		MoveL Tr_meulage_motif_1_P35,[12.5,500,0,0],z0,Tool \wobj:=Wobj_Part_0;
		MoveL Tr_meulage_motif_1_P36,[12.5,500,0,0],z0,Tool \wobj:=Wobj_Part_0;
		MoveL Tr_meulage_motif_1_P37,[12.5,500,0,0],z0,Tool \wobj:=Wobj_Part_0;
		MoveL Tr_meulage_motif_1_P38,[12.5,500,0,0],z0,Tool \wobj:=Wobj_Part_0;
		MoveL Tr_meulage_motif_1_P39,[12.5,500,0,0],z0,Tool \wobj:=Wobj_Part_0;
		MoveL Tr_meulage_motif_1_P40,[12.5,500,0,0],z0,Tool \wobj:=Wobj_Part_0;
		MoveL Tr_meulage_motif_1_P41,[12.5,500,0,0],z0,Tool \wobj:=Wobj_Part_0;
		MoveL Tr_meulage_motif_1_P42,[12.5,500,0,0],z0,Tool \wobj:=Wobj_Part_0;
		MoveL Tr_meulage_motif_1_P43,[12.5,500,0,0],z0,Tool \wobj:=Wobj_Part_0;
		MoveL Tr_meulage_motif_1_P44,[12.5,500,0,0],z0,Tool \wobj:=Wobj_Part_0;
		MoveL Tr_meulage_motif_1_P45,[12.5,500,0,0],z0,Tool \wobj:=Wobj_Part_0;
		MoveL Tr_meulage_motif_1_P46,[12.5,500,0,0],z0,Tool \wobj:=Wobj_Part_0;
		MoveL Tr_meulage_motif_1_P47,[12.5,500,0,0],z0,Tool \wobj:=Wobj_Part_0;
		MoveL Tr_meulage_motif_1_P48,[12.5,500,0,0],z0,Tool \wobj:=Wobj_Part_0;
		MoveL Tr_meulage_motif_1_P49,[12.5,500,0,0],z0,Tool \wobj:=Wobj_Part_0;
		MoveL Tr_meulage_motif_1_P50,[12.5,500,0,0],z0,Tool \wobj:=Wobj_Part_0;
		MoveL Tr_meulage_motif_1_P51,[12.5,500,0,0],z0,Tool \wobj:=Wobj_Part_0;
		MoveL Tr_meulage_motif_1_P52,[12.5,500,0,0],z0,Tool \wobj:=Wobj_Part_0;
		MoveL Tr_meulage_motif_1_P53,[12.5,500,0,0],z0,Tool \wobj:=Wobj_Part_0;
		MoveL Tr_meulage_motif_1_P54,[12.5,500,0,0],z0,Tool \wobj:=Wobj_Part_0;
		MoveL Tr_meulage_motif_1_P55,[12.5,500,0,0],z0,Tool \wobj:=Wobj_Part_0;
		MoveL Tr_meulage_motif_1_P56,[12.5,500,0,0],z0,Tool \wobj:=Wobj_Part_0;
		MoveL Tr_meulage_motif_1_P57,[12.5,500,0,0],z0,Tool \wobj:=Wobj_Part_0;
		MoveL Tr_meulage_motif_1_P58,[12.5,500,0,0],z0,Tool \wobj:=Wobj_Part_0;
		MoveL Tr_meulage_motif_1_P59,[12.5,500,0,0],z0,Tool \wobj:=Wobj_Part_0;
		MoveL Tr_meulage_motif_1_P60,[12.5,500,0,0],z0,Tool \wobj:=Wobj_Part_0;
		MoveL Tr_meulage_motif_1_P61,[12.5,500,0,0],z0,Tool \wobj:=Wobj_Part_0;
		MoveL Tr_meulage_motif_1_P62,[12.5,500,0,0],z0,Tool \wobj:=Wobj_Part_0;
		MoveL Tr_meulage_motif_1_P63,[12.5,500,0,0],z0,Tool \wobj:=Wobj_Part_0;
		MoveL Tr_meulage_motif_1_P64,[12.5,500,0,0],z0,Tool \wobj:=Wobj_Part_0;
		MoveL Tr_meulage_motif_1_P65,[12.5,500,0,0],z0,Tool \wobj:=Wobj_Part_0;
		MoveL Tr_meulage_motif_1_P66,[12.5,500,0,0],z0,Tool \wobj:=Wobj_Part_0;
		MoveL Tr_meulage_motif_1_P67,[12.5,500,0,0],z0,Tool \wobj:=Wobj_Part_0;
		MoveL Tr_meulage_motif_1_P68,[12.5,500,0,0],z0,Tool \wobj:=Wobj_Part_0;
		MoveL Tr_meulage_motif_1_P69,[12.5,500,0,0],z0,Tool \wobj:=Wobj_Part_0;
		MoveL Tr_meulage_motif_1_P70,[12.5,500,0,0],z0,Tool \wobj:=Wobj_Part_0;
		MoveL Tr_meulage_motif_1_P71,[12.5,500,0,0],z0,Tool \wobj:=Wobj_Part_0;
		MoveL Tr_meulage_motif_1_P72,[12.5,500,0,0],z0,Tool \wobj:=Wobj_Part_0;
		MoveL Tr_meulage_motif_1_P73,[12.5,500,0,0],z0,Tool \wobj:=Wobj_Part_0;
		MoveL Tr_meulage_motif_1_P74,[12.5,500,0,0],z0,Tool \wobj:=Wobj_Part_0;
		MoveL Tr_meulage_motif_1_P75,[12.5,500,0,0],z0,Tool \wobj:=Wobj_Part_0;
		MoveL Tr_meulage_motif_1_P76,[12.5,500,0,0],z0,Tool \wobj:=Wobj_Part_0;
		MoveL Tr_meulage_motif_1_P77,[12.5,500,0,0],z0,Tool \wobj:=Wobj_Part_0;
		MoveL Tr_meulage_motif_1_P78,[12.5,500,0,0],z0,Tool \wobj:=Wobj_Part_0;
		MoveL Tr_meulage_motif_1_P79,[12.5,500,0,0],z0,Tool \wobj:=Wobj_Part_0;
		MoveL Tr_meulage_motif_1_P80,[12.5,500,0,0],z0,Tool \wobj:=Wobj_Part_0;
		MoveL Tr_meulage_motif_1_P81,[12.5,500,0,0],z0,Tool \wobj:=Wobj_Part_0;
		MoveL Tr_meulage_motif_1_P82,[12.5,500,0,0],z0,Tool \wobj:=Wobj_Part_0;
		MoveL Tr_meulage_motif_1_P83,[12.5,500,0,0],z0,Tool \wobj:=Wobj_Part_0;
		MoveL Tr_meulage_motif_1_P84,[12.5,500,0,0],z0,Tool \wobj:=Wobj_Part_0;
		MoveL Tr_meulage_motif_1_P85,[12.5,500,0,0],z0,Tool \wobj:=Wobj_Part_0;
		MoveL Tr_meulage_motif_1_P86,[12.5,500,0,0],z0,Tool \wobj:=Wobj_Part_0;
		MoveL Tr_meulage_motif_1_P87,[12.5,500,0,0],z0,Tool \wobj:=Wobj_Part_0;
		MoveL Tr_meulage_motif_1_P88,[12.5,500,0,0],z0,Tool \wobj:=Wobj_Part_0;
		MoveL Tr_meulage_motif_1_P89,[12.5,500,0,0],z0,Tool \wobj:=Wobj_Part_0;
		MoveL Tr_meulage_motif_1_P90,[12.5,500,0,0],z0,Tool \wobj:=Wobj_Part_0;
		MoveL Tr_meulage_motif_1_P91,[12.5,500,0,0],z0,Tool \wobj:=Wobj_Part_0;
		MoveL Tr_meulage_motif_1_P92,[12.5,500,0,0],z0,Tool \wobj:=Wobj_Part_0;
		MoveL Tr_meulage_motif_1_P93,[12.5,500,0,0],z0,Tool \wobj:=Wobj_Part_0;
		MoveL Tr_meulage_motif_1_P94,[12.5,500,0,0],z0,Tool \wobj:=Wobj_Part_0;
		MoveL Tr_meulage_motif_1_P95,[12.5,500,0,0],z0,Tool \wobj:=Wobj_Part_0;
		MoveL Tr_meulage_motif_1_P96,[12.5,500,0,0],z0,Tool \wobj:=Wobj_Part_0;
		MoveL Tr_meulage_motif_1_P97,[12.5,500,0,0],z0,Tool \wobj:=Wobj_Part_0;
		MoveL Tr_meulage_motif_1_P98,[12.5,500,0,0],z0,Tool \wobj:=Wobj_Part_0;
		MoveL Tr_meulage_motif_1_P99,[12.5,500,0,0],z0,Tool \wobj:=Wobj_Part_0;
		MoveL Tr_meulage_motif_1_P100,[12.5,500,0,0],z0,Tool \wobj:=Wobj_Part_0;
		MoveL Tr_meulage_motif_1_P101,[12.5,500,0,0],z0,Tool \wobj:=Wobj_Part_0;
		MoveL Tr_meulage_motif_1_P102,[12.5,500,0,0],z0,Tool \wobj:=Wobj_Part_0;
		MoveL Tr_meulage_motif_1_P103,[12.5,500,0,0],z0,Tool \wobj:=Wobj_Part_0;
		MoveL Tr_meulage_motif_1_P104,[12.5,500,0,0],z0,Tool \wobj:=Wobj_Part_0;
		MoveL Tr_meulage_motif_1_P105,[12.5,500,0,0],z0,Tool \wobj:=Wobj_Part_0;
		MoveL Tr_meulage_motif_1_P106,[12.5,500,0,0],z0,Tool \wobj:=Wobj_Part_0;
		MoveL Tr_meulage_motif_1_P107,[12.5,500,0,0],z0,Tool \wobj:=Wobj_Part_0;
		MoveL Tr_meulage_motif_1_P108,[12.5,500,0,0],z0,Tool \wobj:=Wobj_Part_0;
		MoveL Tr_meulage_motif_1_P109,[12.5,500,0,0],z0,Tool \wobj:=Wobj_Part_0;
		MoveL Tr_meulage_motif_1_P110,[12.5,500,0,0],z0,Tool \wobj:=Wobj_Part_0;
		MoveL Tr_meulage_motif_1_P111,[12.5,500,0,0],z0,Tool \wobj:=Wobj_Part_0;
		MoveL Tr_meulage_motif_1_P112,[12.5,500,0,0],z0,Tool \wobj:=Wobj_Part_0;
		MoveL Tr_meulage_motif_1_P113,[12.5,500,0,0],z0,Tool \wobj:=Wobj_Part_0;
		MoveL Tr_meulage_motif_1_P114,[12.5,500,0,0],z0,Tool \wobj:=Wobj_Part_0;
		MoveL Tr_meulage_motif_1_P115,[12.5,500,0,0],z0,Tool \wobj:=Wobj_Part_0;
		MoveJ Tr_meulage_motif_1_degg1,V500,Z0,Tool,\Wobj:=Wobj_Part_0;
		MoveJ Tr_meulage_motif_1_degg2,V2000,Z100,Tool,\Wobj:=Wobj_Part_0;
	ENDPROC
	LOCAL PROC Tr_meulage_motif_2()
		!!Programme Tr_meulage_motif_2 - 24/03/2023 10:23:34;
		 CONST Speeddata vitesse_Meulage :=[50, 500, 0, 0];
		confJ \off;
		confL \off;
		Tool := ToolOffset(Tool_M1_D500_S270);
		MoveAbsJ [[0,-40,40,0,90,0],[8.999999E+09,8.999999E+09,8.999999E+09,8.999999E+09,8.999999E+09,8.999999E+09]] ,V1000,Z0,Tool_M1_D500_S270 \Wobj:=Wobj_Part_0;
		MoveJ Tr_meulage_motif_2_App1,V2000,Z100,Tool,\Wobj:=Wobj_Part_0;
		MoveJ Tr_meulage_motif_2_App2,V500,Z0,Tool,\Wobj:=Wobj_Part_0;
		MoveL Tr_meulage_motif_2_P0,[12.5,500,0,0],z0,Tool \wobj:=Wobj_Part_0;
		MoveL Tr_meulage_motif_2_P1,[12.5,500,0,0],z0,Tool \wobj:=Wobj_Part_0;
		MoveL Tr_meulage_motif_2_P2,[12.5,500,0,0],z0,Tool \wobj:=Wobj_Part_0;
		MoveL Tr_meulage_motif_2_P3,[12.5,500,0,0],z0,Tool \wobj:=Wobj_Part_0;
		MoveL Tr_meulage_motif_2_P4,[12.5,500,0,0],z0,Tool \wobj:=Wobj_Part_0;
		MoveL Tr_meulage_motif_2_P5,[12.5,500,0,0],z0,Tool \wobj:=Wobj_Part_0;
		MoveL Tr_meulage_motif_2_P6,[12.5,500,0,0],z0,Tool \wobj:=Wobj_Part_0;
		MoveL Tr_meulage_motif_2_P7,[12.5,500,0,0],z0,Tool \wobj:=Wobj_Part_0;
		MoveL Tr_meulage_motif_2_P8,[12.5,500,0,0],z0,Tool \wobj:=Wobj_Part_0;
		MoveL Tr_meulage_motif_2_P9,[12.5,500,0,0],z0,Tool \wobj:=Wobj_Part_0;
		MoveL Tr_meulage_motif_2_P10,[12.5,500,0,0],z0,Tool \wobj:=Wobj_Part_0;
		MoveL Tr_meulage_motif_2_P11,[12.5,500,0,0],z0,Tool \wobj:=Wobj_Part_0;
		MoveL Tr_meulage_motif_2_P12,[12.5,500,0,0],z0,Tool \wobj:=Wobj_Part_0;
		MoveL Tr_meulage_motif_2_P13,[12.5,500,0,0],z0,Tool \wobj:=Wobj_Part_0;
		MoveL Tr_meulage_motif_2_P14,[12.5,500,0,0],z0,Tool \wobj:=Wobj_Part_0;
		MoveL Tr_meulage_motif_2_P15,[12.5,500,0,0],z0,Tool \wobj:=Wobj_Part_0;
		MoveL Tr_meulage_motif_2_P16,[12.5,500,0,0],z0,Tool \wobj:=Wobj_Part_0;
		MoveL Tr_meulage_motif_2_P17,[12.5,500,0,0],z0,Tool \wobj:=Wobj_Part_0;
		MoveL Tr_meulage_motif_2_P18,[12.5,500,0,0],z0,Tool \wobj:=Wobj_Part_0;
		MoveL Tr_meulage_motif_2_P19,[12.5,500,0,0],z0,Tool \wobj:=Wobj_Part_0;
		MoveL Tr_meulage_motif_2_P20,[12.5,500,0,0],z0,Tool \wobj:=Wobj_Part_0;
		MoveL Tr_meulage_motif_2_P21,[12.5,500,0,0],z0,Tool \wobj:=Wobj_Part_0;
		MoveL Tr_meulage_motif_2_P22,[12.5,500,0,0],z0,Tool \wobj:=Wobj_Part_0;
		MoveL Tr_meulage_motif_2_P23,[12.5,500,0,0],z0,Tool \wobj:=Wobj_Part_0;
		MoveL Tr_meulage_motif_2_P24,[12.5,500,0,0],z0,Tool \wobj:=Wobj_Part_0;
		MoveL Tr_meulage_motif_2_P25,[12.5,500,0,0],z0,Tool \wobj:=Wobj_Part_0;
		MoveL Tr_meulage_motif_2_P26,[12.5,500,0,0],z0,Tool \wobj:=Wobj_Part_0;
		MoveL Tr_meulage_motif_2_P27,[12.5,500,0,0],z0,Tool \wobj:=Wobj_Part_0;
		MoveL Tr_meulage_motif_2_P28,[12.5,500,0,0],z0,Tool \wobj:=Wobj_Part_0;
		MoveL Tr_meulage_motif_2_P29,[12.5,500,0,0],z0,Tool \wobj:=Wobj_Part_0;
		MoveL Tr_meulage_motif_2_P30,[12.5,500,0,0],z0,Tool \wobj:=Wobj_Part_0;
		MoveL Tr_meulage_motif_2_P31,[12.5,500,0,0],z0,Tool \wobj:=Wobj_Part_0;
		MoveL Tr_meulage_motif_2_P32,[12.5,500,0,0],z0,Tool \wobj:=Wobj_Part_0;
		MoveL Tr_meulage_motif_2_P33,[12.5,500,0,0],z0,Tool \wobj:=Wobj_Part_0;
		MoveL Tr_meulage_motif_2_P34,[12.5,500,0,0],z0,Tool \wobj:=Wobj_Part_0;
		MoveL Tr_meulage_motif_2_P35,[12.5,500,0,0],z0,Tool \wobj:=Wobj_Part_0;
		MoveL Tr_meulage_motif_2_P36,[12.5,500,0,0],z0,Tool \wobj:=Wobj_Part_0;
		MoveL Tr_meulage_motif_2_P37,[12.5,500,0,0],z0,Tool \wobj:=Wobj_Part_0;
		MoveL Tr_meulage_motif_2_P38,[12.5,500,0,0],z0,Tool \wobj:=Wobj_Part_0;
		MoveL Tr_meulage_motif_2_P39,[12.5,500,0,0],z0,Tool \wobj:=Wobj_Part_0;
		MoveL Tr_meulage_motif_2_P40,[12.5,500,0,0],z0,Tool \wobj:=Wobj_Part_0;
		MoveL Tr_meulage_motif_2_P41,[12.5,500,0,0],z0,Tool \wobj:=Wobj_Part_0;
		MoveL Tr_meulage_motif_2_P42,[12.5,500,0,0],z0,Tool \wobj:=Wobj_Part_0;
		MoveL Tr_meulage_motif_2_P43,[12.5,500,0,0],z0,Tool \wobj:=Wobj_Part_0;
		MoveL Tr_meulage_motif_2_P44,[12.5,500,0,0],z0,Tool \wobj:=Wobj_Part_0;
		MoveL Tr_meulage_motif_2_P45,[12.5,500,0,0],z0,Tool \wobj:=Wobj_Part_0;
		MoveL Tr_meulage_motif_2_P46,[12.5,500,0,0],z0,Tool \wobj:=Wobj_Part_0;
		MoveL Tr_meulage_motif_2_P47,[12.5,500,0,0],z0,Tool \wobj:=Wobj_Part_0;
		MoveL Tr_meulage_motif_2_P48,[12.5,500,0,0],z0,Tool \wobj:=Wobj_Part_0;
		MoveL Tr_meulage_motif_2_P49,[12.5,500,0,0],z0,Tool \wobj:=Wobj_Part_0;
		MoveL Tr_meulage_motif_2_P50,[12.5,500,0,0],z0,Tool \wobj:=Wobj_Part_0;
		MoveL Tr_meulage_motif_2_P51,[12.5,500,0,0],z0,Tool \wobj:=Wobj_Part_0;
		MoveL Tr_meulage_motif_2_P52,[12.5,500,0,0],z0,Tool \wobj:=Wobj_Part_0;
		MoveL Tr_meulage_motif_2_P53,[12.5,500,0,0],z0,Tool \wobj:=Wobj_Part_0;
		MoveL Tr_meulage_motif_2_P54,[12.5,500,0,0],z0,Tool \wobj:=Wobj_Part_0;
		MoveL Tr_meulage_motif_2_P55,[12.5,500,0,0],z0,Tool \wobj:=Wobj_Part_0;
		MoveL Tr_meulage_motif_2_P56,[12.5,500,0,0],z0,Tool \wobj:=Wobj_Part_0;
		MoveL Tr_meulage_motif_2_P57,[12.5,500,0,0],z0,Tool \wobj:=Wobj_Part_0;
		MoveL Tr_meulage_motif_2_P58,[12.5,500,0,0],z0,Tool \wobj:=Wobj_Part_0;
		MoveL Tr_meulage_motif_2_P59,[12.5,500,0,0],z0,Tool \wobj:=Wobj_Part_0;
		MoveL Tr_meulage_motif_2_P60,[12.5,500,0,0],z0,Tool \wobj:=Wobj_Part_0;
		MoveL Tr_meulage_motif_2_P61,[12.5,500,0,0],z0,Tool \wobj:=Wobj_Part_0;
		MoveL Tr_meulage_motif_2_P62,[12.5,500,0,0],z0,Tool \wobj:=Wobj_Part_0;
		MoveL Tr_meulage_motif_2_P63,[12.5,500,0,0],z0,Tool \wobj:=Wobj_Part_0;
		MoveL Tr_meulage_motif_2_P64,[12.5,500,0,0],z0,Tool \wobj:=Wobj_Part_0;
		MoveL Tr_meulage_motif_2_P65,[12.5,500,0,0],z0,Tool \wobj:=Wobj_Part_0;
		MoveL Tr_meulage_motif_2_P66,[12.5,500,0,0],z0,Tool \wobj:=Wobj_Part_0;
		MoveL Tr_meulage_motif_2_P67,[12.5,500,0,0],z0,Tool \wobj:=Wobj_Part_0;
		MoveL Tr_meulage_motif_2_P68,[12.5,500,0,0],z0,Tool \wobj:=Wobj_Part_0;
		MoveL Tr_meulage_motif_2_P69,[12.5,500,0,0],z0,Tool \wobj:=Wobj_Part_0;
		MoveL Tr_meulage_motif_2_P70,[12.5,500,0,0],z0,Tool \wobj:=Wobj_Part_0;
		MoveL Tr_meulage_motif_2_P71,[12.5,500,0,0],z0,Tool \wobj:=Wobj_Part_0;
		MoveL Tr_meulage_motif_2_P72,[12.5,500,0,0],z0,Tool \wobj:=Wobj_Part_0;
		MoveL Tr_meulage_motif_2_P73,[12.5,500,0,0],z0,Tool \wobj:=Wobj_Part_0;
		MoveL Tr_meulage_motif_2_P74,[12.5,500,0,0],z0,Tool \wobj:=Wobj_Part_0;
		MoveL Tr_meulage_motif_2_P75,[12.5,500,0,0],z0,Tool \wobj:=Wobj_Part_0;
		MoveL Tr_meulage_motif_2_P76,[12.5,500,0,0],z0,Tool \wobj:=Wobj_Part_0;
		MoveL Tr_meulage_motif_2_P77,[12.5,500,0,0],z0,Tool \wobj:=Wobj_Part_0;
		MoveL Tr_meulage_motif_2_P78,[12.5,500,0,0],z0,Tool \wobj:=Wobj_Part_0;
		MoveL Tr_meulage_motif_2_P79,[12.5,500,0,0],z0,Tool \wobj:=Wobj_Part_0;
		MoveL Tr_meulage_motif_2_P80,[12.5,500,0,0],z0,Tool \wobj:=Wobj_Part_0;
		MoveL Tr_meulage_motif_2_P81,[12.5,500,0,0],z0,Tool \wobj:=Wobj_Part_0;
		MoveL Tr_meulage_motif_2_P82,[12.5,500,0,0],z0,Tool \wobj:=Wobj_Part_0;
		MoveL Tr_meulage_motif_2_P83,[12.5,500,0,0],z0,Tool \wobj:=Wobj_Part_0;
		MoveL Tr_meulage_motif_2_P84,[12.5,500,0,0],z0,Tool \wobj:=Wobj_Part_0;
		MoveL Tr_meulage_motif_2_P85,[12.5,500,0,0],z0,Tool \wobj:=Wobj_Part_0;
		MoveL Tr_meulage_motif_2_P86,[12.5,500,0,0],z0,Tool \wobj:=Wobj_Part_0;
		MoveL Tr_meulage_motif_2_P87,[12.5,500,0,0],z0,Tool \wobj:=Wobj_Part_0;
		MoveL Tr_meulage_motif_2_P88,[12.5,500,0,0],z0,Tool \wobj:=Wobj_Part_0;
		MoveL Tr_meulage_motif_2_P89,[12.5,500,0,0],z0,Tool \wobj:=Wobj_Part_0;
		MoveL Tr_meulage_motif_2_P90,[12.5,500,0,0],z0,Tool \wobj:=Wobj_Part_0;
		MoveL Tr_meulage_motif_2_P91,[12.5,500,0,0],z0,Tool \wobj:=Wobj_Part_0;
		MoveL Tr_meulage_motif_2_P92,[12.5,500,0,0],z0,Tool \wobj:=Wobj_Part_0;
		MoveL Tr_meulage_motif_2_P93,[12.5,500,0,0],z0,Tool \wobj:=Wobj_Part_0;
		MoveL Tr_meulage_motif_2_P94,[12.5,500,0,0],z0,Tool \wobj:=Wobj_Part_0;
		MoveL Tr_meulage_motif_2_P95,[12.5,500,0,0],z0,Tool \wobj:=Wobj_Part_0;
		MoveL Tr_meulage_motif_2_P96,[12.5,500,0,0],z0,Tool \wobj:=Wobj_Part_0;
		MoveL Tr_meulage_motif_2_P97,[12.5,500,0,0],z0,Tool \wobj:=Wobj_Part_0;
		MoveL Tr_meulage_motif_2_P98,[12.5,500,0,0],z0,Tool \wobj:=Wobj_Part_0;
		MoveL Tr_meulage_motif_2_P99,[12.5,500,0,0],z0,Tool \wobj:=Wobj_Part_0;
		MoveL Tr_meulage_motif_2_P100,[12.5,500,0,0],z0,Tool \wobj:=Wobj_Part_0;
		MoveL Tr_meulage_motif_2_P101,[12.5,500,0,0],z0,Tool \wobj:=Wobj_Part_0;
		MoveL Tr_meulage_motif_2_P102,[12.5,500,0,0],z0,Tool \wobj:=Wobj_Part_0;
		MoveL Tr_meulage_motif_2_P103,[12.5,500,0,0],z0,Tool \wobj:=Wobj_Part_0;
		MoveL Tr_meulage_motif_2_P104,[12.5,500,0,0],z0,Tool \wobj:=Wobj_Part_0;
		MoveL Tr_meulage_motif_2_P105,[12.5,500,0,0],z0,Tool \wobj:=Wobj_Part_0;
		MoveL Tr_meulage_motif_2_P106,[12.5,500,0,0],z0,Tool \wobj:=Wobj_Part_0;
		MoveL Tr_meulage_motif_2_P107,[12.5,500,0,0],z0,Tool \wobj:=Wobj_Part_0;
		MoveL Tr_meulage_motif_2_P108,[12.5,500,0,0],z0,Tool \wobj:=Wobj_Part_0;
		MoveL Tr_meulage_motif_2_P109,[12.5,500,0,0],z0,Tool \wobj:=Wobj_Part_0;
		MoveL Tr_meulage_motif_2_P110,[12.5,500,0,0],z0,Tool \wobj:=Wobj_Part_0;
		MoveL Tr_meulage_motif_2_P111,[12.5,500,0,0],z0,Tool \wobj:=Wobj_Part_0;
		MoveL Tr_meulage_motif_2_P112,[12.5,500,0,0],z0,Tool \wobj:=Wobj_Part_0;
		MoveL Tr_meulage_motif_2_P113,[12.5,500,0,0],z0,Tool \wobj:=Wobj_Part_0;
		MoveL Tr_meulage_motif_2_P114,[12.5,500,0,0],z0,Tool \wobj:=Wobj_Part_0;
		MoveL Tr_meulage_motif_2_P115,[12.5,500,0,0],z0,Tool \wobj:=Wobj_Part_0;
		MoveJ Tr_meulage_motif_2_degg1,V500,Z0,Tool,\Wobj:=Wobj_Part_0;
		MoveJ Tr_meulage_motif_2_degg2,V2000,Z100,Tool,\Wobj:=Wobj_Part_0;
	ENDPROC
	LOCAL PROC Tr_meulage_bavure()
		!!Programme Tr_meulage_bavure - 24/03/2023 10:23:34;
		 CONST Speeddata vitesse_Meulage :=[50, 500, 0, 0];
		confJ \off;
		confL \off;
		Tool := ToolOffset(Tool_M1_D500_S0);
		MoveAbsJ [[0,-40,40,0,90,0],[8.999999E+09,8.999999E+09,8.999999E+09,8.999999E+09,8.999999E+09,8.999999E+09]] ,V1000,Z0,Tool_M1_D500_S0 \Wobj:=Wobj_Part_0;
		MoveJ Tr_meulage_bavure_App1,V2000,Z100,Tool,\Wobj:=Wobj_Part_0;
		MoveJ Tr_meulage_bavure_App2,V500,Z0,Tool,\Wobj:=Wobj_Part_0;
		MoveL Tr_meulage_bavure_P0,[50,500,0,0],z0,Tool \wobj:=Wobj_Part_0;
		MoveL Tr_meulage_bavure_P1,[50,500,0,0],z0,Tool \wobj:=Wobj_Part_0;
		MoveL Tr_meulage_bavure_P2,[50,500,0,0],z0,Tool \wobj:=Wobj_Part_0;
		MoveL Tr_meulage_bavure_P3,[50,500,0,0],z0,Tool \wobj:=Wobj_Part_0;
		MoveL Tr_meulage_bavure_P4,[50,500,0,0],z0,Tool \wobj:=Wobj_Part_0;
		MoveL Tr_meulage_bavure_P5,[50,500,0,0],z0,Tool \wobj:=Wobj_Part_0;
		MoveL Tr_meulage_bavure_P6,[50,500,0,0],z0,Tool \wobj:=Wobj_Part_0;
		MoveL Tr_meulage_bavure_P7,[50,500,0,0],z0,Tool \wobj:=Wobj_Part_0;
		MoveL Tr_meulage_bavure_P8,[50,500,0,0],z0,Tool \wobj:=Wobj_Part_0;
		MoveL Tr_meulage_bavure_P9,[50,500,0,0],z0,Tool \wobj:=Wobj_Part_0;
		MoveL Tr_meulage_bavure_P10,[50,500,0,0],z0,Tool \wobj:=Wobj_Part_0;
		MoveL Tr_meulage_bavure_P11,[50,500,0,0],z0,Tool \wobj:=Wobj_Part_0;
		MoveL Tr_meulage_bavure_P12,[50,500,0,0],z0,Tool \wobj:=Wobj_Part_0;
		MoveL Tr_meulage_bavure_P13,[50,500,0,0],z0,Tool \wobj:=Wobj_Part_0;
		MoveL Tr_meulage_bavure_P14,[50,500,0,0],z0,Tool \wobj:=Wobj_Part_0;
		MoveL Tr_meulage_bavure_P15,[50,500,0,0],z0,Tool \wobj:=Wobj_Part_0;
		MoveL Tr_meulage_bavure_P16,[50,500,0,0],z0,Tool \wobj:=Wobj_Part_0;
		MoveL Tr_meulage_bavure_P17,[50,500,0,0],z0,Tool \wobj:=Wobj_Part_0;
		MoveL Tr_meulage_bavure_P18,[50,500,0,0],z0,Tool \wobj:=Wobj_Part_0;
		MoveL Tr_meulage_bavure_P19,[50,500,0,0],z0,Tool \wobj:=Wobj_Part_0;
		MoveL Tr_meulage_bavure_P20,[50,500,0,0],z0,Tool \wobj:=Wobj_Part_0;
		MoveL Tr_meulage_bavure_P21,[50,500,0,0],z0,Tool \wobj:=Wobj_Part_0;
		MoveL Tr_meulage_bavure_P22,[50,500,0,0],z0,Tool \wobj:=Wobj_Part_0;
		MoveL Tr_meulage_bavure_P23,[50,500,0,0],z0,Tool \wobj:=Wobj_Part_0;
		MoveL Tr_meulage_bavure_P24,[50,500,0,0],z0,Tool \wobj:=Wobj_Part_0;
		MoveL Tr_meulage_bavure_P25,[50,500,0,0],z0,Tool \wobj:=Wobj_Part_0;
		MoveL Tr_meulage_bavure_P26,[50,500,0,0],z0,Tool \wobj:=Wobj_Part_0;
		MoveL Tr_meulage_bavure_P27,[50,500,0,0],z0,Tool \wobj:=Wobj_Part_0;
		MoveL Tr_meulage_bavure_P28,[50,500,0,0],z0,Tool \wobj:=Wobj_Part_0;
		MoveL Tr_meulage_bavure_P29,[50,500,0,0],z0,Tool \wobj:=Wobj_Part_0;
		MoveL Tr_meulage_bavure_P30,[50,500,0,0],z0,Tool \wobj:=Wobj_Part_0;
		MoveL Tr_meulage_bavure_P31,[50,500,0,0],z0,Tool \wobj:=Wobj_Part_0;
		MoveL Tr_meulage_bavure_P32,[50,500,0,0],z0,Tool \wobj:=Wobj_Part_0;
		MoveL Tr_meulage_bavure_P33,[50,500,0,0],z0,Tool \wobj:=Wobj_Part_0;
		MoveL Tr_meulage_bavure_P34,[50,500,0,0],z0,Tool \wobj:=Wobj_Part_0;
		MoveL Tr_meulage_bavure_P35,[50,500,0,0],z0,Tool \wobj:=Wobj_Part_0;
		MoveL Tr_meulage_bavure_P36,[50,500,0,0],z0,Tool \wobj:=Wobj_Part_0;
		MoveL Tr_meulage_bavure_P37,[50,500,0,0],z0,Tool \wobj:=Wobj_Part_0;
		MoveL Tr_meulage_bavure_P38,[50,500,0,0],z0,Tool \wobj:=Wobj_Part_0;
		MoveL Tr_meulage_bavure_P39,[50,500,0,0],z0,Tool \wobj:=Wobj_Part_0;
		MoveL Tr_meulage_bavure_P40,[50,500,0,0],z0,Tool \wobj:=Wobj_Part_0;
		MoveL Tr_meulage_bavure_P41,[50,500,0,0],z0,Tool \wobj:=Wobj_Part_0;
		MoveL Tr_meulage_bavure_P42,[50,500,0,0],z0,Tool \wobj:=Wobj_Part_0;
		MoveL Tr_meulage_bavure_P43,[50,500,0,0],z0,Tool \wobj:=Wobj_Part_0;
		MoveL Tr_meulage_bavure_P44,[50,500,0,0],z0,Tool \wobj:=Wobj_Part_0;
		MoveL Tr_meulage_bavure_P45,[50,500,0,0],z0,Tool \wobj:=Wobj_Part_0;
		MoveL Tr_meulage_bavure_P46,[50,500,0,0],z0,Tool \wobj:=Wobj_Part_0;
		MoveL Tr_meulage_bavure_P47,[50,500,0,0],z0,Tool \wobj:=Wobj_Part_0;
		MoveL Tr_meulage_bavure_P48,[50,500,0,0],z0,Tool \wobj:=Wobj_Part_0;
		MoveL Tr_meulage_bavure_P49,[50,500,0,0],z0,Tool \wobj:=Wobj_Part_0;
		MoveL Tr_meulage_bavure_P50,[50,500,0,0],z0,Tool \wobj:=Wobj_Part_0;
		MoveL Tr_meulage_bavure_P51,[50,500,0,0],z0,Tool \wobj:=Wobj_Part_0;
		MoveL Tr_meulage_bavure_P52,[50,500,0,0],z0,Tool \wobj:=Wobj_Part_0;
		MoveL Tr_meulage_bavure_P53,[50,500,0,0],z0,Tool \wobj:=Wobj_Part_0;
		MoveL Tr_meulage_bavure_P54,[50,500,0,0],z0,Tool \wobj:=Wobj_Part_0;
		MoveL Tr_meulage_bavure_P55,[50,500,0,0],z0,Tool \wobj:=Wobj_Part_0;
		MoveL Tr_meulage_bavure_P56,[50,500,0,0],z0,Tool \wobj:=Wobj_Part_0;
		MoveL Tr_meulage_bavure_P57,[50,500,0,0],z0,Tool \wobj:=Wobj_Part_0;
		MoveL Tr_meulage_bavure_P58,[50,500,0,0],z0,Tool \wobj:=Wobj_Part_0;
		MoveL Tr_meulage_bavure_P59,[50,500,0,0],z0,Tool \wobj:=Wobj_Part_0;
		MoveL Tr_meulage_bavure_P60,[50,500,0,0],z0,Tool \wobj:=Wobj_Part_0;
		MoveL Tr_meulage_bavure_P61,[50,500,0,0],z0,Tool \wobj:=Wobj_Part_0;
		MoveL Tr_meulage_bavure_P62,[50,500,0,0],z0,Tool \wobj:=Wobj_Part_0;
		MoveL Tr_meulage_bavure_P63,[50,500,0,0],z0,Tool \wobj:=Wobj_Part_0;
		MoveL Tr_meulage_bavure_P64,[50,500,0,0],z0,Tool \wobj:=Wobj_Part_0;
		MoveL Tr_meulage_bavure_P65,[50,500,0,0],z0,Tool \wobj:=Wobj_Part_0;
		MoveL Tr_meulage_bavure_P66,[50,500,0,0],z0,Tool \wobj:=Wobj_Part_0;
		MoveL Tr_meulage_bavure_P67,[50,500,0,0],z0,Tool \wobj:=Wobj_Part_0;
		MoveL Tr_meulage_bavure_P68,[50,500,0,0],z0,Tool \wobj:=Wobj_Part_0;
		MoveL Tr_meulage_bavure_P69,[50,500,0,0],z0,Tool \wobj:=Wobj_Part_0;
		MoveL Tr_meulage_bavure_P70,[50,500,0,0],z0,Tool \wobj:=Wobj_Part_0;
		MoveL Tr_meulage_bavure_P71,[50,500,0,0],z0,Tool \wobj:=Wobj_Part_0;
		MoveL Tr_meulage_bavure_P72,[50,500,0,0],z0,Tool \wobj:=Wobj_Part_0;
		MoveL Tr_meulage_bavure_P73,[50,500,0,0],z0,Tool \wobj:=Wobj_Part_0;
		MoveL Tr_meulage_bavure_P74,[50,500,0,0],z0,Tool \wobj:=Wobj_Part_0;
		MoveL Tr_meulage_bavure_P75,[50,500,0,0],z0,Tool \wobj:=Wobj_Part_0;
		MoveL Tr_meulage_bavure_P76,[50,500,0,0],z0,Tool \wobj:=Wobj_Part_0;
		MoveL Tr_meulage_bavure_P77,[50,500,0,0],z0,Tool \wobj:=Wobj_Part_0;
		MoveL Tr_meulage_bavure_P78,[50,500,0,0],z0,Tool \wobj:=Wobj_Part_0;
		MoveL Tr_meulage_bavure_P79,[50,500,0,0],z0,Tool \wobj:=Wobj_Part_0;
		MoveL Tr_meulage_bavure_P80,[50,500,0,0],z0,Tool \wobj:=Wobj_Part_0;
		MoveL Tr_meulage_bavure_P81,[50,500,0,0],z0,Tool \wobj:=Wobj_Part_0;
		MoveL Tr_meulage_bavure_P82,[50,500,0,0],z0,Tool \wobj:=Wobj_Part_0;
		MoveL Tr_meulage_bavure_P83,[50,500,0,0],z0,Tool \wobj:=Wobj_Part_0;
		MoveL Tr_meulage_bavure_P84,[50,500,0,0],z0,Tool \wobj:=Wobj_Part_0;
		MoveL Tr_meulage_bavure_P85,[50,500,0,0],z0,Tool \wobj:=Wobj_Part_0;
		MoveL Tr_meulage_bavure_P86,[50,500,0,0],z0,Tool \wobj:=Wobj_Part_0;
		MoveL Tr_meulage_bavure_P87,[50,500,0,0],z0,Tool \wobj:=Wobj_Part_0;
		MoveL Tr_meulage_bavure_P88,[50,500,0,0],z0,Tool \wobj:=Wobj_Part_0;
		MoveL Tr_meulage_bavure_P89,[50,500,0,0],z0,Tool \wobj:=Wobj_Part_0;
		MoveL Tr_meulage_bavure_P90,[50,500,0,0],z0,Tool \wobj:=Wobj_Part_0;
		MoveL Tr_meulage_bavure_P91,[50,500,0,0],z0,Tool \wobj:=Wobj_Part_0;
		MoveL Tr_meulage_bavure_P92,[50,500,0,0],z0,Tool \wobj:=Wobj_Part_0;
		MoveL Tr_meulage_bavure_P93,[50,500,0,0],z0,Tool \wobj:=Wobj_Part_0;
		MoveL Tr_meulage_bavure_P94,[50,500,0,0],z0,Tool \wobj:=Wobj_Part_0;
		MoveL Tr_meulage_bavure_P95,[50,500,0,0],z0,Tool \wobj:=Wobj_Part_0;
		MoveL Tr_meulage_bavure_P96,[50,500,0,0],z0,Tool \wobj:=Wobj_Part_0;
		MoveL Tr_meulage_bavure_P97,[50,500,0,0],z0,Tool \wobj:=Wobj_Part_0;
		MoveL Tr_meulage_bavure_P98,[50,500,0,0],z0,Tool \wobj:=Wobj_Part_0;
		MoveL Tr_meulage_bavure_P99,[50,500,0,0],z0,Tool \wobj:=Wobj_Part_0;
		MoveL Tr_meulage_bavure_P100,[50,500,0,0],z0,Tool \wobj:=Wobj_Part_0;
		MoveL Tr_meulage_bavure_P101,[50,500,0,0],z0,Tool \wobj:=Wobj_Part_0;
		MoveL Tr_meulage_bavure_P102,[50,500,0,0],z0,Tool \wobj:=Wobj_Part_0;
		MoveL Tr_meulage_bavure_P103,[50,500,0,0],z0,Tool \wobj:=Wobj_Part_0;
		MoveL Tr_meulage_bavure_P104,[50,500,0,0],z0,Tool \wobj:=Wobj_Part_0;
		MoveL Tr_meulage_bavure_P105,[50,500,0,0],z0,Tool \wobj:=Wobj_Part_0;
		MoveL Tr_meulage_bavure_P106,[50,500,0,0],z0,Tool \wobj:=Wobj_Part_0;
		MoveL Tr_meulage_bavure_P107,[50,500,0,0],z0,Tool \wobj:=Wobj_Part_0;
		MoveL Tr_meulage_bavure_P108,[50,500,0,0],z0,Tool \wobj:=Wobj_Part_0;
		MoveL Tr_meulage_bavure_P109,[50,500,0,0],z0,Tool \wobj:=Wobj_Part_0;
		MoveL Tr_meulage_bavure_P110,[50,500,0,0],z0,Tool \wobj:=Wobj_Part_0;
		MoveL Tr_meulage_bavure_P111,[50,500,0,0],z0,Tool \wobj:=Wobj_Part_0;
		MoveL Tr_meulage_bavure_P112,[50,500,0,0],z0,Tool \wobj:=Wobj_Part_0;
		MoveL Tr_meulage_bavure_P113,[50,500,0,0],z0,Tool \wobj:=Wobj_Part_0;
		MoveL Tr_meulage_bavure_P114,[50,500,0,0],z0,Tool \wobj:=Wobj_Part_0;
		MoveL Tr_meulage_bavure_P115,[50,500,0,0],z0,Tool \wobj:=Wobj_Part_0;
		MoveL Tr_meulage_bavure_P116,[50,500,0,0],z0,Tool \wobj:=Wobj_Part_0;
		MoveL Tr_meulage_bavure_P117,[50,500,0,0],z0,Tool \wobj:=Wobj_Part_0;
		MoveL Tr_meulage_bavure_P118,[50,500,0,0],z0,Tool \wobj:=Wobj_Part_0;
		MoveL Tr_meulage_bavure_P119,[50,500,0,0],z0,Tool \wobj:=Wobj_Part_0;
		MoveL Tr_meulage_bavure_P120,[50,500,0,0],z0,Tool \wobj:=Wobj_Part_0;
		MoveL Tr_meulage_bavure_P121,[50,500,0,0],z0,Tool \wobj:=Wobj_Part_0;
		MoveL Tr_meulage_bavure_P122,[50,500,0,0],z0,Tool \wobj:=Wobj_Part_0;
		MoveL Tr_meulage_bavure_P123,[50,500,0,0],z0,Tool \wobj:=Wobj_Part_0;
		MoveL Tr_meulage_bavure_P124,[50,500,0,0],z0,Tool \wobj:=Wobj_Part_0;
		MoveL Tr_meulage_bavure_P125,[50,500,0,0],z0,Tool \wobj:=Wobj_Part_0;
		MoveL Tr_meulage_bavure_P126,[50,500,0,0],z0,Tool \wobj:=Wobj_Part_0;
		MoveL Tr_meulage_bavure_P127,[50,500,0,0],z0,Tool \wobj:=Wobj_Part_0;
		MoveL Tr_meulage_bavure_P128,[50,500,0,0],z0,Tool \wobj:=Wobj_Part_0;
		MoveL Tr_meulage_bavure_P129,[50,500,0,0],z0,Tool \wobj:=Wobj_Part_0;
		MoveL Tr_meulage_bavure_P130,[50,500,0,0],z0,Tool \wobj:=Wobj_Part_0;
		MoveL Tr_meulage_bavure_P131,[50,500,0,0],z0,Tool \wobj:=Wobj_Part_0;
		MoveL Tr_meulage_bavure_P132,[50,500,0,0],z0,Tool \wobj:=Wobj_Part_0;
		MoveL Tr_meulage_bavure_P133,[50,500,0,0],z0,Tool \wobj:=Wobj_Part_0;
		MoveL Tr_meulage_bavure_P134,[50,500,0,0],z0,Tool \wobj:=Wobj_Part_0;
		MoveL Tr_meulage_bavure_P135,[50,500,0,0],z0,Tool \wobj:=Wobj_Part_0;
		MoveL Tr_meulage_bavure_P136,[50,500,0,0],z0,Tool \wobj:=Wobj_Part_0;
		MoveL Tr_meulage_bavure_P137,[50,500,0,0],z0,Tool \wobj:=Wobj_Part_0;
		MoveL Tr_meulage_bavure_P138,[50,500,0,0],z0,Tool \wobj:=Wobj_Part_0;
		MoveL Tr_meulage_bavure_P139,[50,500,0,0],z0,Tool \wobj:=Wobj_Part_0;
		MoveL Tr_meulage_bavure_P140,[50,500,0,0],z0,Tool \wobj:=Wobj_Part_0;
		MoveL Tr_meulage_bavure_P141,[50,500,0,0],z0,Tool \wobj:=Wobj_Part_0;
		MoveL Tr_meulage_bavure_P142,[50,500,0,0],z0,Tool \wobj:=Wobj_Part_0;
		MoveL Tr_meulage_bavure_P143,[50,500,0,0],z0,Tool \wobj:=Wobj_Part_0;
		MoveL Tr_meulage_bavure_P144,[50,500,0,0],z0,Tool \wobj:=Wobj_Part_0;
		MoveL Tr_meulage_bavure_P145,[50,500,0,0],z0,Tool \wobj:=Wobj_Part_0;
		MoveL Tr_meulage_bavure_P146,[50,500,0,0],z0,Tool \wobj:=Wobj_Part_0;
		MoveL Tr_meulage_bavure_P147,[50,500,0,0],z0,Tool \wobj:=Wobj_Part_0;
		MoveL Tr_meulage_bavure_P148,[50,500,0,0],z0,Tool \wobj:=Wobj_Part_0;
		MoveL Tr_meulage_bavure_P149,[50,500,0,0],z0,Tool \wobj:=Wobj_Part_0;
		MoveL Tr_meulage_bavure_P150,[50,500,0,0],z0,Tool \wobj:=Wobj_Part_0;
		MoveL Tr_meulage_bavure_P151,[50,500,0,0],z0,Tool \wobj:=Wobj_Part_0;
		MoveL Tr_meulage_bavure_P152,[50,500,0,0],z0,Tool \wobj:=Wobj_Part_0;
		MoveL Tr_meulage_bavure_P153,[50,500,0,0],z0,Tool \wobj:=Wobj_Part_0;
		MoveL Tr_meulage_bavure_P154,[50,500,0,0],z0,Tool \wobj:=Wobj_Part_0;
		MoveL Tr_meulage_bavure_P155,[50,500,0,0],z0,Tool \wobj:=Wobj_Part_0;
		MoveL Tr_meulage_bavure_P156,[50,500,0,0],z0,Tool \wobj:=Wobj_Part_0;
		MoveL Tr_meulage_bavure_P157,[50,500,0,0],z0,Tool \wobj:=Wobj_Part_0;
		MoveL Tr_meulage_bavure_P158,[50,500,0,0],z0,Tool \wobj:=Wobj_Part_0;
		MoveL Tr_meulage_bavure_P159,[50,500,0,0],z0,Tool \wobj:=Wobj_Part_0;
		MoveL Tr_meulage_bavure_P160,[50,500,0,0],z0,Tool \wobj:=Wobj_Part_0;
		MoveL Tr_meulage_bavure_P161,[50,500,0,0],z0,Tool \wobj:=Wobj_Part_0;
		MoveL Tr_meulage_bavure_P162,[50,500,0,0],z0,Tool \wobj:=Wobj_Part_0;
		MoveL Tr_meulage_bavure_P163,[50,500,0,0],z0,Tool \wobj:=Wobj_Part_0;
		MoveL Tr_meulage_bavure_P164,[50,500,0,0],z0,Tool \wobj:=Wobj_Part_0;
		MoveL Tr_meulage_bavure_P165,[50,500,0,0],z0,Tool \wobj:=Wobj_Part_0;
		MoveL Tr_meulage_bavure_P166,[50,500,0,0],z0,Tool \wobj:=Wobj_Part_0;
		MoveL Tr_meulage_bavure_P167,[50,500,0,0],z0,Tool \wobj:=Wobj_Part_0;
		MoveL Tr_meulage_bavure_P168,[50,500,0,0],z0,Tool \wobj:=Wobj_Part_0;
		MoveL Tr_meulage_bavure_P169,[50,500,0,0],z0,Tool \wobj:=Wobj_Part_0;
		MoveL Tr_meulage_bavure_P170,[50,500,0,0],z0,Tool \wobj:=Wobj_Part_0;
		MoveL Tr_meulage_bavure_P171,[50,500,0,0],z0,Tool \wobj:=Wobj_Part_0;
		MoveL Tr_meulage_bavure_P172,[50,500,0,0],z0,Tool \wobj:=Wobj_Part_0;
		MoveL Tr_meulage_bavure_P173,[50,500,0,0],z0,Tool \wobj:=Wobj_Part_0;
		MoveL Tr_meulage_bavure_P174,[50,500,0,0],z0,Tool \wobj:=Wobj_Part_0;
		MoveL Tr_meulage_bavure_P175,[50,500,0,0],z0,Tool \wobj:=Wobj_Part_0;
		MoveL Tr_meulage_bavure_P176,[50,500,0,0],z0,Tool \wobj:=Wobj_Part_0;
		MoveL Tr_meulage_bavure_P177,[50,500,0,0],z0,Tool \wobj:=Wobj_Part_0;
		MoveL Tr_meulage_bavure_P178,[50,500,0,0],z0,Tool \wobj:=Wobj_Part_0;
		MoveL Tr_meulage_bavure_P179,[50,500,0,0],z0,Tool \wobj:=Wobj_Part_0;
		MoveL Tr_meulage_bavure_P180,[50,500,0,0],z0,Tool \wobj:=Wobj_Part_0;
		MoveL Tr_meulage_bavure_P181,[50,500,0,0],z0,Tool \wobj:=Wobj_Part_0;
		MoveL Tr_meulage_bavure_P182,[50,500,0,0],z0,Tool \wobj:=Wobj_Part_0;
		MoveL Tr_meulage_bavure_P183,[50,500,0,0],z0,Tool \wobj:=Wobj_Part_0;
		MoveL Tr_meulage_bavure_P184,[50,500,0,0],z0,Tool \wobj:=Wobj_Part_0;
		MoveL Tr_meulage_bavure_P185,[50,500,0,0],z0,Tool \wobj:=Wobj_Part_0;
		MoveL Tr_meulage_bavure_P186,[50,500,0,0],z0,Tool \wobj:=Wobj_Part_0;
		MoveL Tr_meulage_bavure_P187,[50,500,0,0],z0,Tool \wobj:=Wobj_Part_0;
		MoveL Tr_meulage_bavure_P188,[50,500,0,0],z0,Tool \wobj:=Wobj_Part_0;
		MoveL Tr_meulage_bavure_P189,[50,500,0,0],z0,Tool \wobj:=Wobj_Part_0;
		MoveL Tr_meulage_bavure_P190,[50,500,0,0],z0,Tool \wobj:=Wobj_Part_0;
		MoveL Tr_meulage_bavure_P191,[50,500,0,0],z0,Tool \wobj:=Wobj_Part_0;
		MoveL Tr_meulage_bavure_P192,[50,500,0,0],z0,Tool \wobj:=Wobj_Part_0;
		MoveL Tr_meulage_bavure_P193,[50,500,0,0],z0,Tool \wobj:=Wobj_Part_0;
		MoveL Tr_meulage_bavure_P194,[50,500,0,0],z0,Tool \wobj:=Wobj_Part_0;
		MoveL Tr_meulage_bavure_P195,[50,500,0,0],z0,Tool \wobj:=Wobj_Part_0;
		MoveL Tr_meulage_bavure_P196,[50,500,0,0],z0,Tool \wobj:=Wobj_Part_0;
		MoveL Tr_meulage_bavure_P197,[50,500,0,0],z0,Tool \wobj:=Wobj_Part_0;
		MoveL Tr_meulage_bavure_P198,[50,500,0,0],z0,Tool \wobj:=Wobj_Part_0;
		MoveL Tr_meulage_bavure_P199,[50,500,0,0],z0,Tool \wobj:=Wobj_Part_0;
		MoveL Tr_meulage_bavure_P200,[50,500,0,0],z0,Tool \wobj:=Wobj_Part_0;
		MoveL Tr_meulage_bavure_P201,[50,500,0,0],z0,Tool \wobj:=Wobj_Part_0;
		MoveL Tr_meulage_bavure_P202,[50,500,0,0],z0,Tool \wobj:=Wobj_Part_0;
		MoveL Tr_meulage_bavure_P203,[50,500,0,0],z0,Tool \wobj:=Wobj_Part_0;
		MoveL Tr_meulage_bavure_P204,[50,500,0,0],z0,Tool \wobj:=Wobj_Part_0;
		MoveL Tr_meulage_bavure_P205,[50,500,0,0],z0,Tool \wobj:=Wobj_Part_0;
		MoveL Tr_meulage_bavure_P206,[50,500,0,0],z0,Tool \wobj:=Wobj_Part_0;
		MoveL Tr_meulage_bavure_P207,[50,500,0,0],z0,Tool \wobj:=Wobj_Part_0;
		MoveL Tr_meulage_bavure_P208,[50,500,0,0],z0,Tool \wobj:=Wobj_Part_0;
		MoveL Tr_meulage_bavure_P209,[50,500,0,0],z0,Tool \wobj:=Wobj_Part_0;
		MoveL Tr_meulage_bavure_P210,[50,500,0,0],z0,Tool \wobj:=Wobj_Part_0;
		MoveL Tr_meulage_bavure_P211,[50,500,0,0],z0,Tool \wobj:=Wobj_Part_0;
		MoveL Tr_meulage_bavure_P212,[50,500,0,0],z0,Tool \wobj:=Wobj_Part_0;
		MoveL Tr_meulage_bavure_P213,[50,500,0,0],z0,Tool \wobj:=Wobj_Part_0;
		MoveL Tr_meulage_bavure_P214,[50,500,0,0],z0,Tool \wobj:=Wobj_Part_0;
		MoveL Tr_meulage_bavure_P215,[50,500,0,0],z0,Tool \wobj:=Wobj_Part_0;
		MoveL Tr_meulage_bavure_P216,[50,500,0,0],z0,Tool \wobj:=Wobj_Part_0;
		MoveL Tr_meulage_bavure_P217,[50,500,0,0],z0,Tool \wobj:=Wobj_Part_0;
		MoveL Tr_meulage_bavure_P218,[50,500,0,0],z0,Tool \wobj:=Wobj_Part_0;
		MoveL Tr_meulage_bavure_P219,[50,500,0,0],z0,Tool \wobj:=Wobj_Part_0;
		MoveL Tr_meulage_bavure_P220,[50,500,0,0],z0,Tool \wobj:=Wobj_Part_0;
		MoveL Tr_meulage_bavure_P221,[50,500,0,0],z0,Tool \wobj:=Wobj_Part_0;
		MoveL Tr_meulage_bavure_P222,[50,500,0,0],z0,Tool \wobj:=Wobj_Part_0;
		MoveL Tr_meulage_bavure_P223,[50,500,0,0],z0,Tool \wobj:=Wobj_Part_0;
		MoveL Tr_meulage_bavure_P224,[50,500,0,0],z0,Tool \wobj:=Wobj_Part_0;
		MoveL Tr_meulage_bavure_P225,[50,500,0,0],z0,Tool \wobj:=Wobj_Part_0;
		MoveL Tr_meulage_bavure_P226,[50,500,0,0],z0,Tool \wobj:=Wobj_Part_0;
		MoveL Tr_meulage_bavure_P227,[50,500,0,0],z0,Tool \wobj:=Wobj_Part_0;
		MoveL Tr_meulage_bavure_P228,[50,500,0,0],z0,Tool \wobj:=Wobj_Part_0;
		MoveL Tr_meulage_bavure_P229,[50,500,0,0],z0,Tool \wobj:=Wobj_Part_0;
		MoveL Tr_meulage_bavure_P230,[50,500,0,0],z0,Tool \wobj:=Wobj_Part_0;
		MoveL Tr_meulage_bavure_P231,[50,500,0,0],z0,Tool \wobj:=Wobj_Part_0;
		MoveL Tr_meulage_bavure_P232,[50,500,0,0],z0,Tool \wobj:=Wobj_Part_0;
		MoveL Tr_meulage_bavure_P233,[50,500,0,0],z0,Tool \wobj:=Wobj_Part_0;
		MoveL Tr_meulage_bavure_P234,[50,500,0,0],z0,Tool \wobj:=Wobj_Part_0;
		MoveL Tr_meulage_bavure_P235,[50,500,0,0],z0,Tool \wobj:=Wobj_Part_0;
		MoveL Tr_meulage_bavure_P236,[50,500,0,0],z0,Tool \wobj:=Wobj_Part_0;
		MoveL Tr_meulage_bavure_P237,[50,500,0,0],z0,Tool \wobj:=Wobj_Part_0;
		MoveL Tr_meulage_bavure_P238,[50,500,0,0],z0,Tool \wobj:=Wobj_Part_0;
		MoveL Tr_meulage_bavure_P239,[50,500,0,0],z0,Tool \wobj:=Wobj_Part_0;
		MoveL Tr_meulage_bavure_P240,[50,500,0,0],z0,Tool \wobj:=Wobj_Part_0;
		MoveL Tr_meulage_bavure_P241,[50,500,0,0],z0,Tool \wobj:=Wobj_Part_0;
		MoveL Tr_meulage_bavure_P242,[50,500,0,0],z0,Tool \wobj:=Wobj_Part_0;
		MoveL Tr_meulage_bavure_P243,[50,500,0,0],z0,Tool \wobj:=Wobj_Part_0;
		MoveL Tr_meulage_bavure_P244,[50,500,0,0],z0,Tool \wobj:=Wobj_Part_0;
		MoveL Tr_meulage_bavure_P245,[50,500,0,0],z0,Tool \wobj:=Wobj_Part_0;
		MoveL Tr_meulage_bavure_P246,[50,500,0,0],z0,Tool \wobj:=Wobj_Part_0;
		MoveL Tr_meulage_bavure_P247,[50,500,0,0],z0,Tool \wobj:=Wobj_Part_0;
		MoveL Tr_meulage_bavure_P248,[50,500,0,0],z0,Tool \wobj:=Wobj_Part_0;
		MoveL Tr_meulage_bavure_P249,[50,500,0,0],z0,Tool \wobj:=Wobj_Part_0;
		MoveL Tr_meulage_bavure_P250,[50,500,0,0],z0,Tool \wobj:=Wobj_Part_0;
		MoveL Tr_meulage_bavure_P251,[50,500,0,0],z0,Tool \wobj:=Wobj_Part_0;
		MoveL Tr_meulage_bavure_P252,[50,500,0,0],z0,Tool \wobj:=Wobj_Part_0;
		MoveL Tr_meulage_bavure_P253,[50,500,0,0],z0,Tool \wobj:=Wobj_Part_0;
		MoveL Tr_meulage_bavure_P254,[50,500,0,0],z0,Tool \wobj:=Wobj_Part_0;
		MoveL Tr_meulage_bavure_P255,[50,500,0,0],z0,Tool \wobj:=Wobj_Part_0;
		MoveL Tr_meulage_bavure_P256,[50,500,0,0],z0,Tool \wobj:=Wobj_Part_0;
		MoveL Tr_meulage_bavure_P257,[50,500,0,0],z0,Tool \wobj:=Wobj_Part_0;
		MoveL Tr_meulage_bavure_P258,[50,500,0,0],z0,Tool \wobj:=Wobj_Part_0;
		MoveL Tr_meulage_bavure_P259,[50,500,0,0],z0,Tool \wobj:=Wobj_Part_0;
		MoveL Tr_meulage_bavure_P260,[50,500,0,0],z0,Tool \wobj:=Wobj_Part_0;
		MoveL Tr_meulage_bavure_P261,[50,500,0,0],z0,Tool \wobj:=Wobj_Part_0;
		MoveL Tr_meulage_bavure_P262,[50,500,0,0],z0,Tool \wobj:=Wobj_Part_0;
		MoveL Tr_meulage_bavure_P263,[50,500,0,0],z0,Tool \wobj:=Wobj_Part_0;
		MoveL Tr_meulage_bavure_P264,[50,500,0,0],z0,Tool \wobj:=Wobj_Part_0;
		MoveL Tr_meulage_bavure_P265,[50,500,0,0],z0,Tool \wobj:=Wobj_Part_0;
		MoveL Tr_meulage_bavure_P266,[50,500,0,0],z0,Tool \wobj:=Wobj_Part_0;
		MoveL Tr_meulage_bavure_P267,[50,500,0,0],z0,Tool \wobj:=Wobj_Part_0;
		MoveL Tr_meulage_bavure_P268,[50,500,0,0],z0,Tool \wobj:=Wobj_Part_0;
		MoveL Tr_meulage_bavure_P269,[50,500,0,0],z0,Tool \wobj:=Wobj_Part_0;
		MoveL Tr_meulage_bavure_P270,[50,500,0,0],z0,Tool \wobj:=Wobj_Part_0;
		MoveL Tr_meulage_bavure_P271,[50,500,0,0],z0,Tool \wobj:=Wobj_Part_0;
		MoveL Tr_meulage_bavure_P272,[50,500,0,0],z0,Tool \wobj:=Wobj_Part_0;
		MoveL Tr_meulage_bavure_P273,[50,500,0,0],z0,Tool \wobj:=Wobj_Part_0;
		MoveL Tr_meulage_bavure_P274,[50,500,0,0],z0,Tool \wobj:=Wobj_Part_0;
		MoveL Tr_meulage_bavure_P275,[50,500,0,0],z0,Tool \wobj:=Wobj_Part_0;
		MoveL Tr_meulage_bavure_P276,[50,500,0,0],z0,Tool \wobj:=Wobj_Part_0;
		MoveL Tr_meulage_bavure_P277,[50,500,0,0],z0,Tool \wobj:=Wobj_Part_0;
		MoveL Tr_meulage_bavure_P278,[50,500,0,0],z0,Tool \wobj:=Wobj_Part_0;
		MoveL Tr_meulage_bavure_P279,[50,500,0,0],z0,Tool \wobj:=Wobj_Part_0;
		MoveL Tr_meulage_bavure_P280,[50,500,0,0],z0,Tool \wobj:=Wobj_Part_0;
		MoveL Tr_meulage_bavure_P281,[50,500,0,0],z0,Tool \wobj:=Wobj_Part_0;
		MoveL Tr_meulage_bavure_P282,[50,500,0,0],z0,Tool \wobj:=Wobj_Part_0;
		MoveL Tr_meulage_bavure_P283,[50,500,0,0],z0,Tool \wobj:=Wobj_Part_0;
		MoveL Tr_meulage_bavure_P284,[50,500,0,0],z0,Tool \wobj:=Wobj_Part_0;
		MoveL Tr_meulage_bavure_P285,[50,500,0,0],z0,Tool \wobj:=Wobj_Part_0;
		MoveL Tr_meulage_bavure_P286,[50,500,0,0],z0,Tool \wobj:=Wobj_Part_0;
		MoveL Tr_meulage_bavure_P287,[50,500,0,0],z0,Tool \wobj:=Wobj_Part_0;
		MoveL Tr_meulage_bavure_P288,[50,500,0,0],z0,Tool \wobj:=Wobj_Part_0;
		MoveL Tr_meulage_bavure_P289,[50,500,0,0],z0,Tool \wobj:=Wobj_Part_0;
		MoveL Tr_meulage_bavure_P290,[50,500,0,0],z0,Tool \wobj:=Wobj_Part_0;
		MoveL Tr_meulage_bavure_P291,[50,500,0,0],z0,Tool \wobj:=Wobj_Part_0;
		MoveL Tr_meulage_bavure_P292,[50,500,0,0],z0,Tool \wobj:=Wobj_Part_0;
		MoveL Tr_meulage_bavure_P293,[50,500,0,0],z0,Tool \wobj:=Wobj_Part_0;
		MoveL Tr_meulage_bavure_P294,[50,500,0,0],z0,Tool \wobj:=Wobj_Part_0;
		MoveL Tr_meulage_bavure_P295,[50,500,0,0],z0,Tool \wobj:=Wobj_Part_0;
		MoveL Tr_meulage_bavure_P296,[50,500,0,0],z0,Tool \wobj:=Wobj_Part_0;
		MoveL Tr_meulage_bavure_P297,[50,500,0,0],z0,Tool \wobj:=Wobj_Part_0;
		MoveL Tr_meulage_bavure_P298,[50,500,0,0],z0,Tool \wobj:=Wobj_Part_0;
		MoveL Tr_meulage_bavure_P299,[50,500,0,0],z0,Tool \wobj:=Wobj_Part_0;
		MoveL Tr_meulage_bavure_P300,[50,500,0,0],z0,Tool \wobj:=Wobj_Part_0;
		MoveL Tr_meulage_bavure_P301,[50,500,0,0],z0,Tool \wobj:=Wobj_Part_0;
		MoveL Tr_meulage_bavure_P302,[50,500,0,0],z0,Tool \wobj:=Wobj_Part_0;
		MoveL Tr_meulage_bavure_P303,[50,500,0,0],z0,Tool \wobj:=Wobj_Part_0;
		MoveL Tr_meulage_bavure_P304,[50,500,0,0],z0,Tool \wobj:=Wobj_Part_0;
		MoveL Tr_meulage_bavure_P305,[50,500,0,0],z0,Tool \wobj:=Wobj_Part_0;
		MoveL Tr_meulage_bavure_P306,[50,500,0,0],z0,Tool \wobj:=Wobj_Part_0;
		MoveL Tr_meulage_bavure_P307,[50,500,0,0],z0,Tool \wobj:=Wobj_Part_0;
		MoveL Tr_meulage_bavure_P308,[50,500,0,0],z0,Tool \wobj:=Wobj_Part_0;
		MoveL Tr_meulage_bavure_P309,[50,500,0,0],z0,Tool \wobj:=Wobj_Part_0;
		MoveL Tr_meulage_bavure_P310,[50,500,0,0],z0,Tool \wobj:=Wobj_Part_0;
		MoveL Tr_meulage_bavure_P311,[50,500,0,0],z0,Tool \wobj:=Wobj_Part_0;
		MoveL Tr_meulage_bavure_P312,[50,500,0,0],z0,Tool \wobj:=Wobj_Part_0;
		MoveL Tr_meulage_bavure_P313,[50,500,0,0],z0,Tool \wobj:=Wobj_Part_0;
		MoveL Tr_meulage_bavure_P314,[50,500,0,0],z0,Tool \wobj:=Wobj_Part_0;
		MoveL Tr_meulage_bavure_P315,[50,500,0,0],z0,Tool \wobj:=Wobj_Part_0;
		MoveL Tr_meulage_bavure_P316,[50,500,0,0],z0,Tool \wobj:=Wobj_Part_0;
		MoveL Tr_meulage_bavure_P317,[50,500,0,0],z0,Tool \wobj:=Wobj_Part_0;
		MoveL Tr_meulage_bavure_P318,[50,500,0,0],z0,Tool \wobj:=Wobj_Part_0;
		MoveL Tr_meulage_bavure_P319,[50,500,0,0],z0,Tool \wobj:=Wobj_Part_0;
		MoveL Tr_meulage_bavure_P320,[50,500,0,0],z0,Tool \wobj:=Wobj_Part_0;
		MoveL Tr_meulage_bavure_P321,[50,500,0,0],z0,Tool \wobj:=Wobj_Part_0;
		MoveL Tr_meulage_bavure_P322,[50,500,0,0],z0,Tool \wobj:=Wobj_Part_0;
		MoveL Tr_meulage_bavure_P323,[50,500,0,0],z0,Tool \wobj:=Wobj_Part_0;
		MoveL Tr_meulage_bavure_P324,[50,500,0,0],z0,Tool \wobj:=Wobj_Part_0;
		MoveL Tr_meulage_bavure_P325,[50,500,0,0],z0,Tool \wobj:=Wobj_Part_0;
		MoveL Tr_meulage_bavure_P326,[50,500,0,0],z0,Tool \wobj:=Wobj_Part_0;
		MoveL Tr_meulage_bavure_P327,[50,500,0,0],z0,Tool \wobj:=Wobj_Part_0;
		MoveL Tr_meulage_bavure_P328,[50,500,0,0],z0,Tool \wobj:=Wobj_Part_0;
		MoveL Tr_meulage_bavure_P329,[50,500,0,0],z0,Tool \wobj:=Wobj_Part_0;
		MoveL Tr_meulage_bavure_P330,[50,500,0,0],z0,Tool \wobj:=Wobj_Part_0;
		MoveL Tr_meulage_bavure_P331,[50,500,0,0],z0,Tool \wobj:=Wobj_Part_0;
		MoveL Tr_meulage_bavure_P332,[50,500,0,0],z0,Tool \wobj:=Wobj_Part_0;
		MoveL Tr_meulage_bavure_P333,[50,500,0,0],z0,Tool \wobj:=Wobj_Part_0;
		MoveL Tr_meulage_bavure_P334,[50,500,0,0],z0,Tool \wobj:=Wobj_Part_0;
		MoveL Tr_meulage_bavure_P335,[50,500,0,0],z0,Tool \wobj:=Wobj_Part_0;
		MoveL Tr_meulage_bavure_P336,[50,500,0,0],z0,Tool \wobj:=Wobj_Part_0;
		MoveL Tr_meulage_bavure_P337,[50,500,0,0],z0,Tool \wobj:=Wobj_Part_0;
		MoveL Tr_meulage_bavure_P338,[50,500,0,0],z0,Tool \wobj:=Wobj_Part_0;
		MoveL Tr_meulage_bavure_P339,[50,500,0,0],z0,Tool \wobj:=Wobj_Part_0;
		MoveL Tr_meulage_bavure_P340,[50,500,0,0],z0,Tool \wobj:=Wobj_Part_0;
		MoveL Tr_meulage_bavure_P341,[50,500,0,0],z0,Tool \wobj:=Wobj_Part_0;
		MoveL Tr_meulage_bavure_P342,[50,500,0,0],z0,Tool \wobj:=Wobj_Part_0;
		MoveL Tr_meulage_bavure_P343,[50,500,0,0],z0,Tool \wobj:=Wobj_Part_0;
		MoveL Tr_meulage_bavure_P344,[50,500,0,0],z0,Tool \wobj:=Wobj_Part_0;
		MoveL Tr_meulage_bavure_P345,[50,500,0,0],z0,Tool \wobj:=Wobj_Part_0;
		MoveL Tr_meulage_bavure_P346,[50,500,0,0],z0,Tool \wobj:=Wobj_Part_0;
		MoveL Tr_meulage_bavure_P347,[50,500,0,0],z0,Tool \wobj:=Wobj_Part_0;
		MoveL Tr_meulage_bavure_P348,[50,500,0,0],z0,Tool \wobj:=Wobj_Part_0;
		MoveL Tr_meulage_bavure_P349,[50,500,0,0],z0,Tool \wobj:=Wobj_Part_0;
		MoveL Tr_meulage_bavure_P350,[50,500,0,0],z0,Tool \wobj:=Wobj_Part_0;
		MoveL Tr_meulage_bavure_P351,[50,500,0,0],z0,Tool \wobj:=Wobj_Part_0;
		MoveL Tr_meulage_bavure_P352,[50,500,0,0],z0,Tool \wobj:=Wobj_Part_0;
		MoveL Tr_meulage_bavure_P353,[50,500,0,0],z0,Tool \wobj:=Wobj_Part_0;
		MoveL Tr_meulage_bavure_P354,[50,500,0,0],z0,Tool \wobj:=Wobj_Part_0;
		MoveL Tr_meulage_bavure_P355,[50,500,0,0],z0,Tool \wobj:=Wobj_Part_0;
		MoveL Tr_meulage_bavure_P356,[50,500,0,0],z0,Tool \wobj:=Wobj_Part_0;
		MoveL Tr_meulage_bavure_P357,[50,500,0,0],z0,Tool \wobj:=Wobj_Part_0;
		MoveL Tr_meulage_bavure_P358,[50,500,0,0],z0,Tool \wobj:=Wobj_Part_0;
		MoveL Tr_meulage_bavure_P359,[50,500,0,0],z0,Tool \wobj:=Wobj_Part_0;
		MoveL Tr_meulage_bavure_P360,[50,500,0,0],z0,Tool \wobj:=Wobj_Part_0;
		MoveL Tr_meulage_bavure_P361,[50,500,0,0],z0,Tool \wobj:=Wobj_Part_0;
		MoveL Tr_meulage_bavure_P362,[50,500,0,0],z0,Tool \wobj:=Wobj_Part_0;
		MoveL Tr_meulage_bavure_P363,[50,500,0,0],z0,Tool \wobj:=Wobj_Part_0;
		MoveL Tr_meulage_bavure_P364,[50,500,0,0],z0,Tool \wobj:=Wobj_Part_0;
		MoveL Tr_meulage_bavure_P365,[50,500,0,0],z0,Tool \wobj:=Wobj_Part_0;
		MoveL Tr_meulage_bavure_P366,[50,500,0,0],z0,Tool \wobj:=Wobj_Part_0;
		MoveL Tr_meulage_bavure_P367,[50,500,0,0],z0,Tool \wobj:=Wobj_Part_0;
		MoveL Tr_meulage_bavure_P368,[50,500,0,0],z0,Tool \wobj:=Wobj_Part_0;
		MoveL Tr_meulage_bavure_P369,[50,500,0,0],z0,Tool \wobj:=Wobj_Part_0;
		MoveL Tr_meulage_bavure_P370,[50,500,0,0],z0,Tool \wobj:=Wobj_Part_0;
		MoveL Tr_meulage_bavure_P371,[50,500,0,0],z0,Tool \wobj:=Wobj_Part_0;
		MoveL Tr_meulage_bavure_P372,[50,500,0,0],z0,Tool \wobj:=Wobj_Part_0;
		MoveL Tr_meulage_bavure_P373,[50,500,0,0],z0,Tool \wobj:=Wobj_Part_0;
		MoveL Tr_meulage_bavure_P374,[50,500,0,0],z0,Tool \wobj:=Wobj_Part_0;
		MoveL Tr_meulage_bavure_P375,[50,500,0,0],z0,Tool \wobj:=Wobj_Part_0;
		MoveL Tr_meulage_bavure_P376,[50,500,0,0],z0,Tool \wobj:=Wobj_Part_0;
		MoveL Tr_meulage_bavure_P377,[50,500,0,0],z0,Tool \wobj:=Wobj_Part_0;
		MoveL Tr_meulage_bavure_P378,[50,500,0,0],z0,Tool \wobj:=Wobj_Part_0;
		MoveL Tr_meulage_bavure_P379,[50,500,0,0],z0,Tool \wobj:=Wobj_Part_0;
		MoveL Tr_meulage_bavure_P380,[50,500,0,0],z0,Tool \wobj:=Wobj_Part_0;
		MoveL Tr_meulage_bavure_P381,[50,500,0,0],z0,Tool \wobj:=Wobj_Part_0;
		MoveL Tr_meulage_bavure_P382,[50,500,0,0],z0,Tool \wobj:=Wobj_Part_0;
		MoveL Tr_meulage_bavure_P383,[50,500,0,0],z0,Tool \wobj:=Wobj_Part_0;
		MoveL Tr_meulage_bavure_P384,[50,500,0,0],z0,Tool \wobj:=Wobj_Part_0;
		MoveL Tr_meulage_bavure_P385,[50,500,0,0],z0,Tool \wobj:=Wobj_Part_0;
		MoveL Tr_meulage_bavure_P386,[50,500,0,0],z0,Tool \wobj:=Wobj_Part_0;
		MoveL Tr_meulage_bavure_P387,[50,500,0,0],z0,Tool \wobj:=Wobj_Part_0;
		MoveL Tr_meulage_bavure_P388,[50,500,0,0],z0,Tool \wobj:=Wobj_Part_0;
		MoveL Tr_meulage_bavure_P389,[50,500,0,0],z0,Tool \wobj:=Wobj_Part_0;
		MoveL Tr_meulage_bavure_P390,[50,500,0,0],z0,Tool \wobj:=Wobj_Part_0;
		MoveL Tr_meulage_bavure_P391,[50,500,0,0],z0,Tool \wobj:=Wobj_Part_0;
		MoveL Tr_meulage_bavure_P392,[50,500,0,0],z0,Tool \wobj:=Wobj_Part_0;
		MoveL Tr_meulage_bavure_P393,[50,500,0,0],z0,Tool \wobj:=Wobj_Part_0;
		MoveL Tr_meulage_bavure_P394,[50,500,0,0],z0,Tool \wobj:=Wobj_Part_0;
		MoveL Tr_meulage_bavure_P395,[50,500,0,0],z0,Tool \wobj:=Wobj_Part_0;
		MoveL Tr_meulage_bavure_P396,[50,500,0,0],z0,Tool \wobj:=Wobj_Part_0;
		MoveL Tr_meulage_bavure_P397,[50,500,0,0],z0,Tool \wobj:=Wobj_Part_0;
		MoveL Tr_meulage_bavure_P398,[50,500,0,0],z0,Tool \wobj:=Wobj_Part_0;
		MoveL Tr_meulage_bavure_P399,[50,500,0,0],z0,Tool \wobj:=Wobj_Part_0;
		MoveL Tr_meulage_bavure_P400,[50,500,0,0],z0,Tool \wobj:=Wobj_Part_0;
		MoveL Tr_meulage_bavure_P401,[50,500,0,0],z0,Tool \wobj:=Wobj_Part_0;
		MoveL Tr_meulage_bavure_P402,[50,500,0,0],z0,Tool \wobj:=Wobj_Part_0;
		MoveL Tr_meulage_bavure_P403,[50,500,0,0],z0,Tool \wobj:=Wobj_Part_0;
		MoveL Tr_meulage_bavure_P404,[50,500,0,0],z0,Tool \wobj:=Wobj_Part_0;
		MoveL Tr_meulage_bavure_P405,[50,500,0,0],z0,Tool \wobj:=Wobj_Part_0;
		MoveL Tr_meulage_bavure_P406,[50,500,0,0],z0,Tool \wobj:=Wobj_Part_0;
		MoveL Tr_meulage_bavure_P407,[50,500,0,0],z0,Tool \wobj:=Wobj_Part_0;
		MoveL Tr_meulage_bavure_P408,[50,500,0,0],z0,Tool \wobj:=Wobj_Part_0;
		MoveL Tr_meulage_bavure_P409,[50,500,0,0],z0,Tool \wobj:=Wobj_Part_0;
		MoveL Tr_meulage_bavure_P410,[50,500,0,0],z0,Tool \wobj:=Wobj_Part_0;
		MoveL Tr_meulage_bavure_P411,[50,500,0,0],z0,Tool \wobj:=Wobj_Part_0;
		MoveL Tr_meulage_bavure_P412,[50,500,0,0],z0,Tool \wobj:=Wobj_Part_0;
		MoveL Tr_meulage_bavure_P413,[50,500,0,0],z0,Tool \wobj:=Wobj_Part_0;
		MoveL Tr_meulage_bavure_P414,[50,500,0,0],z0,Tool \wobj:=Wobj_Part_0;
		MoveL Tr_meulage_bavure_P415,[50,500,0,0],z0,Tool \wobj:=Wobj_Part_0;
		MoveL Tr_meulage_bavure_P416,[50,500,0,0],z0,Tool \wobj:=Wobj_Part_0;
		MoveL Tr_meulage_bavure_P417,[50,500,0,0],z0,Tool \wobj:=Wobj_Part_0;
		MoveL Tr_meulage_bavure_P418,[50,500,0,0],z0,Tool \wobj:=Wobj_Part_0;
		MoveL Tr_meulage_bavure_P419,[50,500,0,0],z0,Tool \wobj:=Wobj_Part_0;
		MoveL Tr_meulage_bavure_P420,[50,500,0,0],z0,Tool \wobj:=Wobj_Part_0;
		MoveL Tr_meulage_bavure_P421,[50,500,0,0],z0,Tool \wobj:=Wobj_Part_0;
		MoveL Tr_meulage_bavure_P422,[50,500,0,0],z0,Tool \wobj:=Wobj_Part_0;
		MoveL Tr_meulage_bavure_P423,[50,500,0,0],z0,Tool \wobj:=Wobj_Part_0;
		MoveL Tr_meulage_bavure_P424,[50,500,0,0],z0,Tool \wobj:=Wobj_Part_0;
		MoveL Tr_meulage_bavure_P425,[50,500,0,0],z0,Tool \wobj:=Wobj_Part_0;
		MoveL Tr_meulage_bavure_P426,[50,500,0,0],z0,Tool \wobj:=Wobj_Part_0;
		MoveL Tr_meulage_bavure_P427,[50,500,0,0],z0,Tool \wobj:=Wobj_Part_0;
		MoveL Tr_meulage_bavure_P428,[50,500,0,0],z0,Tool \wobj:=Wobj_Part_0;
		MoveL Tr_meulage_bavure_P429,[50,500,0,0],z0,Tool \wobj:=Wobj_Part_0;
		MoveL Tr_meulage_bavure_P430,[50,500,0,0],z0,Tool \wobj:=Wobj_Part_0;
		MoveL Tr_meulage_bavure_P431,[50,500,0,0],z0,Tool \wobj:=Wobj_Part_0;
		MoveL Tr_meulage_bavure_P432,[50,500,0,0],z0,Tool \wobj:=Wobj_Part_0;
		MoveL Tr_meulage_bavure_P433,[50,500,0,0],z0,Tool \wobj:=Wobj_Part_0;
		MoveL Tr_meulage_bavure_P434,[50,500,0,0],z0,Tool \wobj:=Wobj_Part_0;
		MoveL Tr_meulage_bavure_P435,[50,500,0,0],z0,Tool \wobj:=Wobj_Part_0;
		MoveL Tr_meulage_bavure_P436,[50,500,0,0],z0,Tool \wobj:=Wobj_Part_0;
		MoveL Tr_meulage_bavure_P437,[50,500,0,0],z0,Tool \wobj:=Wobj_Part_0;
		MoveL Tr_meulage_bavure_P438,[50,500,0,0],z0,Tool \wobj:=Wobj_Part_0;
		MoveL Tr_meulage_bavure_P439,[50,500,0,0],z0,Tool \wobj:=Wobj_Part_0;
		MoveL Tr_meulage_bavure_P440,[50,500,0,0],z0,Tool \wobj:=Wobj_Part_0;
		MoveL Tr_meulage_bavure_P441,[50,500,0,0],z0,Tool \wobj:=Wobj_Part_0;
		MoveL Tr_meulage_bavure_P442,[50,500,0,0],z0,Tool \wobj:=Wobj_Part_0;
		MoveL Tr_meulage_bavure_P443,[50,500,0,0],z0,Tool \wobj:=Wobj_Part_0;
		MoveL Tr_meulage_bavure_P444,[50,500,0,0],z0,Tool \wobj:=Wobj_Part_0;
		MoveL Tr_meulage_bavure_P445,[50,500,0,0],z0,Tool \wobj:=Wobj_Part_0;
		MoveL Tr_meulage_bavure_P446,[50,500,0,0],z0,Tool \wobj:=Wobj_Part_0;
		MoveL Tr_meulage_bavure_P447,[50,500,0,0],z0,Tool \wobj:=Wobj_Part_0;
		MoveL Tr_meulage_bavure_P448,[50,500,0,0],z0,Tool \wobj:=Wobj_Part_0;
		MoveL Tr_meulage_bavure_P449,[50,500,0,0],z0,Tool \wobj:=Wobj_Part_0;
		MoveL Tr_meulage_bavure_P450,[50,500,0,0],z0,Tool \wobj:=Wobj_Part_0;
		MoveL Tr_meulage_bavure_P451,[50,500,0,0],z0,Tool \wobj:=Wobj_Part_0;
		MoveL Tr_meulage_bavure_P452,[50,500,0,0],z0,Tool \wobj:=Wobj_Part_0;
		MoveL Tr_meulage_bavure_P453,[50,500,0,0],z0,Tool \wobj:=Wobj_Part_0;
		MoveL Tr_meulage_bavure_P454,[50,500,0,0],z0,Tool \wobj:=Wobj_Part_0;
		MoveL Tr_meulage_bavure_P455,[50,500,0,0],z0,Tool \wobj:=Wobj_Part_0;
		MoveL Tr_meulage_bavure_P456,[50,500,0,0],z0,Tool \wobj:=Wobj_Part_0;
		MoveL Tr_meulage_bavure_P457,[50,500,0,0],z0,Tool \wobj:=Wobj_Part_0;
		MoveL Tr_meulage_bavure_P458,[50,500,0,0],z0,Tool \wobj:=Wobj_Part_0;
		MoveL Tr_meulage_bavure_P459,[50,500,0,0],z0,Tool \wobj:=Wobj_Part_0;
		MoveL Tr_meulage_bavure_P460,[50,500,0,0],z0,Tool \wobj:=Wobj_Part_0;
		MoveL Tr_meulage_bavure_P461,[50,500,0,0],z0,Tool \wobj:=Wobj_Part_0;
		MoveL Tr_meulage_bavure_P462,[50,500,0,0],z0,Tool \wobj:=Wobj_Part_0;
		MoveL Tr_meulage_bavure_P463,[50,500,0,0],z0,Tool \wobj:=Wobj_Part_0;
		MoveL Tr_meulage_bavure_P464,[50,500,0,0],z0,Tool \wobj:=Wobj_Part_0;
		MoveL Tr_meulage_bavure_P465,[50,500,0,0],z0,Tool \wobj:=Wobj_Part_0;
		MoveL Tr_meulage_bavure_P466,[50,500,0,0],z0,Tool \wobj:=Wobj_Part_0;
		MoveL Tr_meulage_bavure_P467,[50,500,0,0],z0,Tool \wobj:=Wobj_Part_0;
		MoveL Tr_meulage_bavure_P468,[50,500,0,0],z0,Tool \wobj:=Wobj_Part_0;
		MoveL Tr_meulage_bavure_P469,[50,500,0,0],z0,Tool \wobj:=Wobj_Part_0;
		MoveL Tr_meulage_bavure_P470,[50,500,0,0],z0,Tool \wobj:=Wobj_Part_0;
		MoveL Tr_meulage_bavure_P471,[50,500,0,0],z0,Tool \wobj:=Wobj_Part_0;
		MoveL Tr_meulage_bavure_P472,[50,500,0,0],z0,Tool \wobj:=Wobj_Part_0;
		MoveL Tr_meulage_bavure_P473,[50,500,0,0],z0,Tool \wobj:=Wobj_Part_0;
		MoveL Tr_meulage_bavure_P474,[50,500,0,0],z0,Tool \wobj:=Wobj_Part_0;
		MoveL Tr_meulage_bavure_P475,[50,500,0,0],z0,Tool \wobj:=Wobj_Part_0;
		MoveL Tr_meulage_bavure_P476,[50,500,0,0],z0,Tool \wobj:=Wobj_Part_0;
		MoveL Tr_meulage_bavure_P477,[50,500,0,0],z0,Tool \wobj:=Wobj_Part_0;
		MoveL Tr_meulage_bavure_P478,[50,500,0,0],z0,Tool \wobj:=Wobj_Part_0;
		MoveL Tr_meulage_bavure_P479,[50,500,0,0],z0,Tool \wobj:=Wobj_Part_0;
		MoveL Tr_meulage_bavure_P480,[50,500,0,0],z0,Tool \wobj:=Wobj_Part_0;
		MoveL Tr_meulage_bavure_P481,[50,500,0,0],z0,Tool \wobj:=Wobj_Part_0;
		MoveL Tr_meulage_bavure_P482,[50,500,0,0],z0,Tool \wobj:=Wobj_Part_0;
		MoveL Tr_meulage_bavure_P483,[50,500,0,0],z0,Tool \wobj:=Wobj_Part_0;
		MoveL Tr_meulage_bavure_P484,[50,500,0,0],z0,Tool \wobj:=Wobj_Part_0;
		MoveL Tr_meulage_bavure_P485,[50,500,0,0],z0,Tool \wobj:=Wobj_Part_0;
		MoveL Tr_meulage_bavure_P486,[50,500,0,0],z0,Tool \wobj:=Wobj_Part_0;
		MoveL Tr_meulage_bavure_P487,[50,500,0,0],z0,Tool \wobj:=Wobj_Part_0;
		MoveL Tr_meulage_bavure_P488,[50,500,0,0],z0,Tool \wobj:=Wobj_Part_0;
		MoveL Tr_meulage_bavure_P489,[50,500,0,0],z0,Tool \wobj:=Wobj_Part_0;
		MoveL Tr_meulage_bavure_P490,[50,500,0,0],z0,Tool \wobj:=Wobj_Part_0;
		MoveL Tr_meulage_bavure_P491,[50,500,0,0],z0,Tool \wobj:=Wobj_Part_0;
		MoveL Tr_meulage_bavure_P492,[50,500,0,0],z0,Tool \wobj:=Wobj_Part_0;
		MoveL Tr_meulage_bavure_P493,[50,500,0,0],z0,Tool \wobj:=Wobj_Part_0;
		MoveL Tr_meulage_bavure_P494,[50,500,0,0],z0,Tool \wobj:=Wobj_Part_0;
		MoveL Tr_meulage_bavure_P495,[50,500,0,0],z0,Tool \wobj:=Wobj_Part_0;
		MoveL Tr_meulage_bavure_P496,[50,500,0,0],z0,Tool \wobj:=Wobj_Part_0;
		MoveL Tr_meulage_bavure_P497,[50,500,0,0],z0,Tool \wobj:=Wobj_Part_0;
		MoveL Tr_meulage_bavure_P498,[50,500,0,0],z0,Tool \wobj:=Wobj_Part_0;
		MoveL Tr_meulage_bavure_P499,[50,500,0,0],z0,Tool \wobj:=Wobj_Part_0;
		MoveL Tr_meulage_bavure_P500,[50,500,0,0],z0,Tool \wobj:=Wobj_Part_0;
		MoveL Tr_meulage_bavure_P501,[50,500,0,0],z0,Tool \wobj:=Wobj_Part_0;
		MoveL Tr_meulage_bavure_P502,[50,500,0,0],z0,Tool \wobj:=Wobj_Part_0;
		MoveL Tr_meulage_bavure_P503,[50,500,0,0],z0,Tool \wobj:=Wobj_Part_0;
		MoveL Tr_meulage_bavure_P504,[50,500,0,0],z0,Tool \wobj:=Wobj_Part_0;
		MoveL Tr_meulage_bavure_P505,[50,500,0,0],z0,Tool \wobj:=Wobj_Part_0;
		MoveL Tr_meulage_bavure_P506,[50,500,0,0],z0,Tool \wobj:=Wobj_Part_0;
		MoveL Tr_meulage_bavure_P507,[50,500,0,0],z0,Tool \wobj:=Wobj_Part_0;
		MoveL Tr_meulage_bavure_P508,[50,500,0,0],z0,Tool \wobj:=Wobj_Part_0;
		MoveL Tr_meulage_bavure_P509,[50,500,0,0],z0,Tool \wobj:=Wobj_Part_0;
		MoveL Tr_meulage_bavure_P510,[50,500,0,0],z0,Tool \wobj:=Wobj_Part_0;
		MoveL Tr_meulage_bavure_P511,[50,500,0,0],z0,Tool \wobj:=Wobj_Part_0;
		MoveJ Tr_meulage_bavure_degg1,V500,Z0,Tool,\Wobj:=Wobj_Part_0;
		MoveJ Tr_meulage_bavure_degg2,V2000,Z100,Tool,\Wobj:=Wobj_Part_0;
	ENDPROC
	 PROC P90_MAIN()
		Tr_pick;
		Tr_Cut;
		Tr_meulage_motif_1;
		Tr_meulage_motif_2;
		Tr_meulage_bavure;
	ENDPROC
ENDMODULE
